FUNCTION_BLOCK FB_Server
VAR
	_ServerNetID		: T_AmsNetID	:= '';(* TwinCAT TCP/IP server network address *)
	_bEnable			: BOOL 			:= FALSE;(* TRUE => enable server data exchange, FALSE => disable *)
	_bLog			: BOOL 			:= FALSE;(* TRUE => Enable log message output, FALSE => Disable *)
	_sPrefix			: STRING 		:= 'SERVER::';(* Log message description string (allows the identification of log message source) *)
	_eState			: E_SocketConnectionState := eSOCKET_DISCONNECTED;(* TCP/IP connection state *)
	_hServer			: REFERENCE TO T_HSERVER;(* Server connection handle *)
	
	fbConnection	: FB_ServerConnection;(* Server data exchange control function block. Implements one server<->client connection *)
	fbTx 			: FB_FrameFifo;(* Tx fifo *)
	fbRx 			: FB_FrameFifo;(* Rx fifo *)
	fbLog			: FB_LogFifo;(* Log/debug/error fifo *)
	Application : I_Application;
	Initalized: BOOL;
END_VAR

(*-------------------------------- Trigger data exchange -----------------------------------------*)
fbConnection( hServer := _hServer, sSrvNetID := ServerNetID, fbRx := fbRx, fbTx := fbTx, fbLog := fbLog, 
			bEnable := _bEnable, bLog := _bLog, sPrefix := _sPrefix, eState => _eState );
			

			
IF fbConnection.eState = eSOCKET_CONNECTED THEN(* Connection established *)
	(*************************This is depends on application****************************************)
	AppliCation.Receive();
	IF Application.isUpdated THEN
		Application.Send();
	END_IF
	(***********************************************************************************************)
END_IF

METHOD FB_init : BOOL
VAR_INPUT
	bInitRetains : BOOL; // if TRUE, the retain variables are initialized (warm start / cold start)
	bInCopyCode : BOOL;  // if TRUE, the instance afterwards gets moved into the copy code (online change)
	application : I_Application;
END_VAR
THIS^.Application := application;
Init();
END_METHOD

METHOD PRIVATE Init
(* 'REF=' DO NOT WORK IN FB_Init  (Probabaly Bug 4024.53) *)
Application.fbLog REF= fbLog;
Application.fbRx REF= fbRx;
Application.fbTx REF= fbTx;
END_METHOD

PROPERTY isEnabling : BOOL
GET
isEnabling := _bEnable;
END_GET
SET
_bEnable := isEnabling;
END_SET
END_PROPERTY

PROPERTY isLogging : BOOL
GET
isLogging := _bLog;
END_GET
SET
_bLog := isLogging;
END_SET
END_PROPERTY

PROPERTY Name : STRING
GET
Name := _sPrefix;
END_GET
SET
_sPrefix := Name;
END_SET
END_PROPERTY

PROPERTY ServerConnectionHandle : REFERENCE TO T_HSERVER
GET
ServerConnectionHandle REF= _hServer;
END_GET
SET
_hServer REF= ServerConnectionHandle;
END_SET
END_PROPERTY

PROPERTY ServerNetID : T_AmsNetID
GET
ServerNetID := _ServerNetID;
END_GET
SET
_ServerNetID := ServerNetID;
END_SET
END_PROPERTY

PROPERTY State : E_SocketConnectionState
GET
State := _eState;
END_GET
END_PROPERTY

END_FUNCTION_BLOCK

(* stored: Version 1.1.0.1, ProductVersion 3.1.4024.12
   POU FB_Server: Id {e4bb1b20-2692-4ae7-ae7c-c964a0db4aba}, SpecialFunc None
   Method FB_init: Id {5983d63a-b1d4-46de-b4c2-689f20870633}
   Method Init: Id {5c917692-77d0-4b74-a9d1-ad5076ff50e5}
   Property isEnabling: Id {3bd963f5-272d-438f-bc5d-876305915938}
   Get Get: Id {31314264-8d39-4955-9943-81fc1fa890f4}
   Set Set: Id {5eea7aec-b17d-4a7f-98cb-95a2f5e39678}
   Property isLogging: Id {97881ea2-865f-4faa-9f3a-c466add18d92}
   Get Get: Id {03b969f7-8ce5-4787-a3ea-5918bf808469}
   Set Set: Id {a9032657-566d-4af4-81bb-7df6c25a5d45}
   Property Name: Id {1e3cc8af-6a47-4956-a156-f293f3fe3eb0}
   Get Get: Id {f9c5209c-0fc5-4c5f-a9ab-e0ee12b1254b}
   Set Set: Id {db7cf90c-1fd9-4ae4-8969-8bf317d0b17b}
   Property ServerConnectionHandle: Id {beec8623-cf64-4300-939c-58c1e0b8b568}
   Get Get: Id {98038ef6-5ac9-4206-9d18-56808c7a256f}
   Set Set: Id {cc5ab284-8de8-4db9-a158-376a5a44999e}
   Property ServerNetID: Id {7c4d1988-c114-437b-ba34-5545fcd82b1e}
   Get Get: Id {21b440ef-7a01-49f8-a6a4-9d2cf4475ecb}
   Set Set: Id {67043950-9b6d-48d9-b531-9ebf3c4f609f}
   Property State: Id {a8722d75-9c3b-4cea-950b-c3f9150a38ae}
   Get Get: Id {4de26aa8-4d42-4a27-ac2b-585605522b36} *)
